// TwinCAT 3 PLC project PLC1
// ProgramVersion: 3.1.4024.0
// libraries:
//   Tc2_Standard, * (Beckhoff Automation GmbH)
//   Tc2_System, * (Beckhoff Automation GmbH)
//   Tc3_Module, * (Beckhoff Automation GmbH)
// project tree:
//   DUTs/ENUM/ E_RS_Cycle_Stop_Cmds.TcDUT, E_Util_State_Cmd.TcDUT, E_TVSA_Cycles.TcDUT, E_Cluster_State_Cmd.TcDUT, E_Util_Service_Req.TcDUT, E_Util_Service_Sts.TcDUT
//   DUTs/STRUCTS/ ST_RS_SeqNumber.TcDUT, ST_Sequence_Sts.TcDUT, ST_Service_Assigned_Sts.TcDUT, ST_Util_Service_Sts.TcDUT, ST_Util_Service_Req.TcDUT
//   DUTs/UNIONS/ U_SeqStart.TcDUT
//   Functions/ F_Get_Seq_Status.TcPOU
//   Function_Blocks/ FB_Cluster_Control.TcPOU, FB_Service_Dispatcher.TcPOU, FB_ReactorSet.TcPOU, FB_ReactorSet_Control.TcPOU, FB_SetOutput_TwoInputs.TcPOU, FB_Utilities_Control.TcPOU, FB_Utilities_Service.TcPOU, FB_Util_Service_Control.TcPOU
//   GVLs/ CONSTANTS.TcGVL, hmi.TcGVL
//   / PlcTask.TcTTO
//   POUs/ MAIN.TcPOU
// real-time tasks:
//   TASK PlcTask: cycle T#10ms, priority 20, ADS port 350
//   TASK PlcTask1: cycle T#10ms, priority 21, ADS port 351
// I/O:
//   DEVICE Device 1 (EtherCAT Automation Protocol) (disabled), AmsNetId 10.33.70.115.2.1
//     Module1 - Publisher
//     Module1 - Subscriber
// variable links:
//   PLC1/PLC1 Instance <-> Device 1 (EtherCAT Automation Protocol)/Module1 - Publisher
//     PlcTask Outputs/MAIN.cluster_control.fb_rs_control[1].fbRS.out_cooling_pump_sts <-> RS1_Bytes/Outputs/VarData[1]
//     PlcTask Outputs/MAIN.cluster_control.fb_rs_control[1].fbRS.out_cycle_req <-> RS1_Bytes/Outputs/VarData[0]
//     PlcTask Outputs/MAIN.cluster_control.fb_rs_control[1].fbRS.out_deadair_pump_sts <-> RS1_Bytes/Outputs/VarData[2]
//     PlcTask Outputs/MAIN.cluster_control.fb_rs_control[1].fbRS.out_steam_system_sts <-> RS1_Bytes/Outputs/VarData[3]
//   PLC1/PLC1 Instance <-> Device 1 (EtherCAT Automation Protocol)/Module1 - Subscriber
//     PlcTask Inputs/MAIN.cluster_control.fb_rs_control[1].fbRS.in_adsorption_seq_sts <-> RS1_Bytes/Inputs/VarData[0]
//     PlcTask Inputs/MAIN.cluster_control.fb_rs_control[1].fbRS.in_airpress_seq_sts <-> RS1_Bytes/Inputs/VarData[4]
//     PlcTask Inputs/MAIN.cluster_control.fb_rs_control[1].fbRS.in_cooling_seq_sts <-> RS1_Bytes/Inputs/VarData[3]
//     PlcTask Inputs/MAIN.cluster_control.fb_rs_control[1].fbRS.in_desorption_seq_sts <-> RS1_Bytes/Inputs/VarData[2]
//     PlcTask Inputs/MAIN.cluster_control.fb_rs_control[1].fbRS.in_evac_seq_sts <-> RS1_Bytes/Inputs/VarData[1]

CONFIGURATION PLC1
    RESOURCE PLC ON TwinCAT3
        TASK PlcTask(INTERVAL := T#10ms, PRIORITY := 20);
        PROGRAM MAIN WITH PlcTask : MAIN;
    END_RESOURCE
END_CONFIGURATION

// ---- DUTs/ENUM/E_RS_Cycle_Stop_Cmds.TcDUT
{attribute 'qualified_only'}
//{attribute 'strict'}
{attribute 'to_string'}

TYPE E_RS_Cycle_Stop_Cmds :
(
	Clear :=0,
	Stop_Cycle,
	Shutdown_Safe,
	Shutdown_Evac,
	Estop
);
END_TYPE

// ---- DUTs/ENUM/E_Util_State_Cmd.TcDUT
{attribute 'qualified_only'}
//{attribute 'strict'}
{attribute 'to_string'}

TYPE E_Util_State_Cmd :
(
	Idle		:= 0,
	Warmup 		:= 1,
	Activate 	:= 2,
	Shutdown 	:= 3,
	Reset_Fault := 4
);
END_TYPE

// ---- DUTs/ENUM/E_TVSA_Cycles.TcDUT
//{attribute 'qualified_only'}
//{attribute 'strict'}
{attribute 'to_string'}

TYPE E_RS_Cycles :
(
	Idle := 0,
	DeadAirEvac,
	SteamDesorption,
	VacCooling,
	AirRepress,
	Adsorption,
	Estop,
	SafeShutdown,
	Error := 9
);
END_TYPE

// ---- DUTs/ENUM/E_Cluster_State_Cmd.TcDUT
{attribute 'qualified_only'}
//{attribute 'strict'}
{attribute 'to_string'}

TYPE E_Cluster_State_Cmd :
(
	Idle := 0,
	Warmup := 1,
	Cycling := 2,
	Shutdown := 3,
	Reset_Fault := 4
);
END_TYPE

// ---- DUTs/ENUM/E_Util_Service_Req.TcDUT
//{attribute 'qualified_only'}
//{attribute 'strict'}
{attribute 'to_string'}

TYPE E_Util_Service_Req :
(
	Reset_Fault := 0,
	On 			:= 1,
	Off 		:= 2
);
END_TYPE

// ---- DUTs/ENUM/E_Util_Service_Sts.TcDUT
//{attribute 'qualified_only'}
//{attribute 'strict'}
{attribute 'to_string'}

TYPE E_Util_Service_Sts :
(
	PowerUp		:= 0,
	Active		:= 1,
	Running		:= 2,
	Faulted		:= 9
);
END_TYPE

// ---- DUTs/STRUCTS/ST_RS_SeqNumber.TcDUT
{attribute 'qualified_only'}
{attribute 'strict'}
TYPE ST_RS_SeqNumber :
STRUCT
	Idle 			: BIT;
	Adsorption		: BIT;
	DeadAirEvac 	: BIT;
	SteamDesorption : BIT;
	VacCooling		: BIT;
	AirRepress 		: BIT;
	Error 			: BIT;
END_STRUCT
END_TYPE

// ---- DUTs/STRUCTS/ST_Sequence_Sts.TcDUT
TYPE ST_Sequence_Sts :
STRUCT
	not_started : BIT;
	started		: BIT;
	completed	: BIT;
	error		: BIT;
END_STRUCT
END_TYPE

// ---- DUTs/STRUCTS/ST_Service_Assigned_Sts.TcDUT
TYPE ST_Service_Assigned_Sts :
STRUCT
	rs_number : UINT;
	is_assigned : BOOL;
END_STRUCT
END_TYPE

// ---- DUTs/STRUCTS/ST_Util_Service_Sts.TcDUT
TYPE ST_Util_Service_Sts :
STRUCT  
	idle		: BOOL;
	ready 		: BOOL;
	running		: BOOL;
	faulted		: BOOL;
	error_code	: DWORD;
END_STRUCT
END_TYPE

// ---- DUTs/STRUCTS/ST_Util_Service_Req.TcDUT
TYPE ST_Util_Service_Req :
STRUCT
	rs_number 		: UINT;
	request_cmd		: UINT;  // (   0 = release/off , 1 = assign/on , 2 =  reset fault)
END_STRUCT
END_TYPE

// ---- DUTs/UNIONS/U_SeqStart.TcDUT
TYPE U_SeqStart :
UNION
	_seq_st 	: ST_RS_SeqNumber;
	_seq_byte 	: BYTE;
END_UNION
END_TYPE

// ---- GVLs/CONSTANTS.TcGVL

VAR_GLOBAL CONSTANT
	rs_count	: UINT := 6;
END_VAR

// ---- GVLs/hmi.TcGVL
{attribute 'qualified_only'}
VAR_GLOBAL
	// Cluster HMI tags - Commnads/Config
	{attribute 'OPC.UA.DA' := '1'} 
	cluster_auto_mode_cmd				: BOOL;
	{attribute 'OPC.UA.DA' := '1'} 								
	cluster_manual_mode_cmd				: BOOL;
	{attribute 'OPC.UA.DA' := '1'} 
	cluster_state_cmd					: BYTE; 									// 0 = Idle, 1 = warmup, 2 = cycle, 3 = shutdown, 4 = reset_fault
	{attribute 'OPC.UA.DA' := '1'} 
	cluster_rs_select_cmd				: ARRAY [1..rs_count] OF BOOL;  			// rs to be started /stopped
	{attribute 'OPC.UA.DA' := '1'} 
	cluster_rs_stop_cycle_cmd			: INT; 										// 1 = stop cycle, 2 = shutdown safe, 3 = shutdown evac, 4 = estop
	{attribute 'OPC.UA.DA' := '1'}  
	cluster_rs_start_cycle_cmd			: BOOL;										// 1 = start cycle
	{attribute 'OPC.UA.DA' := '1'}  
	cluster_reset_fault_cmd				: BOOL;										// reset cluster fault
	{attribute 'OPC.UA.DA' := '1'} 
	cluster_rs_cycles_cfg				: ARRAY [1..rs_count] OF UINT;  			// cycle to run : 12345 = Full TVSA , 1 = Evac, 2 = Desorp ,3 = Cooling ,4 = Repres ,5 = Adsorp
	{attribute 'OPC.UA.DA' := '1'} 
	clsuter_rs_number_of_cycles_cfg		: ARRAY [1..rs_count] OF UINT;  			// number of cycles to run 
	
	// Cluster HMI Tags - Status
	{attribute 'OPC.UA.DA' := '1'} 
	cluster_rs_control_active_cycle_sts : ARRAY [1..rs_count] OF STRING;
	{attribute 'OPC.UA.DA' := '1'} 
	cluster_active_state_sts			: STRING;

	// Utilities HMI tags
	{attribute 'OPC.UA.DA' := '1'} 
	util_auto_mode_cmd		: BOOL := TRUE;  // TRUE = auto mode, FALSE = manual mode 
	{attribute 'OPC.UA.DA' := '1'}  
	util_cooling_pump_cmd 	: REAL; // 0 = off, 1 = On , 2 = reset_fault
	{attribute 'OPC.UA.DA' := '1'} 
	util_cooling_pump_sts 	: INT;
	{attribute 'OPC.UA.DA' := '1'}  
	util_dead_air_pump_cmd 	: REAL; // 0 = off, 1 = On , 2 = reset_fault
	{attribute 'OPC.UA.DA' := '1'} 
	util_dead_air_pump_sts 	: INT;
	{attribute 'OPC.UA.DA' := '1'}  
	util_steam_system_cmd 	: REAL; // 0 = off, 1 = On , 2 = reset_fault
	{attribute 'OPC.UA.DA' := '1'} 
	util_steam_system_sts 	: INT;
	{attribute 'OPC.UA.DA' := '1'}  
	util_purge_assist_cmd 	: REAL; // 0 = off, 1 = On , 2 = reset_fault
	{attribute 'OPC.UA.DA' := '1'} 
	util_purge_assist_sts 	: INT;
END_VAR

// ---- POUs/MAIN.TcPOU
PROGRAM MAIN
VAR
	cluster_control : FB_Cluster_Control();
	sita_out : REAL;
	sita_in1 : REAL;
	sita_in2 : REAL;
	sita_setout : FB_SetOutput_TwoInputs();
END_VAR

cluster_control();

//sita_out := F_SetOutput_LatestInput(in1 := TO_REAL(sita_in1),in2 := TO_REAL(sita_in2));


sita_setout(io_in1 := sita_in1,io_in2 := sita_in2, o_set_value => sita_out);

END_PROGRAM

// ---- Function_Blocks/FB_Cluster_Control.TcPOU
FUNCTION_BLOCK FB_Cluster_Control
VAR
	fb_rs_control 			: ARRAY[1..rs_count] OF FB_ReactorSet_Control;
	//fb_reactor_set			: ARRAY[1..rs_count] OF FB_ReactorSet;
	rs_error				: BOOL;
	
	fb_utilities_control 	: FB_Utilities_Control;
	
	idx_rs 					: UINT;
	
	{attribute 'to_string'}
	seq_state				: (Idle := 0, Warmup := 1, Ready := 2, Cycling := 3, Shutdown := 4, Error); 
	
	rs_stop_cycle_cmd		: ARRAY[1..rs_count] OF  INT;  
	rs_start_cycle_cmd 		: ARRAY[1..rs_count] OF BOOL;
	
	shutdown_util_cmd		: BOOL;
	
	seq_sts 				: ST_Sequence_Sts;
	
	error_reset_cmd			: BOOL;
	trigger_error_reset		: R_TRIG;
	
	cluster_auto_mode		: BOOL;
END_VAR

// Cluster Shutdown 
IF hmi.cluster_state_cmd = E_Cluster_State_Cmd.Shutdown THEN 
	IF  seq_state =  Cycling AND Get_RS_CycleDone_Sts() THEN 
		seq_state := Shutdown;
	ELSIF seq_state <>  Cycling THEN 
		seq_state := Shutdown;
	END_IF
END_IF


// Cluster States 
CASE seq_state OF 
	
	Idle : 
		fb_utilities_control.i_state_req := E_Cluster_State_Cmd.Idle;
		seq_sts.error := FALSE;
		seq_sts.started := FALSE;
		IF hmi.cluster_state_cmd = E_Cluster_State_Cmd.Warmup THEN 
			seq_sts.completed := FALSE;
			seq_sts.started := TRUE;
			seq_state := Warmup;
		END_IF
		
	Warmup:	
		fb_utilities_control.i_state_req := E_Util_State_Cmd.Warmup;
		IF NOT fb_utilities_control.o_bop_warmup_sts.error  THEN 
			IF fb_utilities_control.o_bop_warmup_sts.completed THEN 
				seq_state := Ready;
			END_IF
		ELSE
			seq_state := Error;
		END_IF		
		
	Ready :
		fb_utilities_control.i_state_req := E_Util_State_Cmd.Activate;
		
		IF  NOT fb_utilities_control.o_bop_error_critical AND NOT rs_error THEN
			IF  fb_utilities_control.o_bop_activate_sts.completed AND hmi.cluster_state_cmd = E_Cluster_State_Cmd.Cycling THEN 
				seq_state := Cycling;
			END_IF
		ELSE
			seq_state := Error;
		END_IF
		
	Cycling :
	
			seq_state := Cycling;
		
	Shutdown : 
		
		fb_utilities_control.i_state_req := E_Util_State_Cmd.Shutdown;
		IF NOT fb_utilities_control.o_bop_shutdown_sts.error THEN 
			IF fb_utilities_control.o_bop_shutdown_sts.completed THEN 
				seq_sts.completed := TRUE;
				seq_state := Idle;
			END_IF
		ELSE
			seq_state := Error;	
		END_IF
	
	Error : 
		seq_sts.completed := TRUE;
		seq_sts.error := TRUE;
		IF error_reset_cmd THEN 
			seq_state := Idle;
		END_IF		
END_CASE


// Reactor Sets and Utilities Cycles Control 
RS_Utilities_Control();

// Error Reset Handling 
Reset_Error();

// ==============  HMI ===================

// HMI auto/manual
IF hmi.cluster_auto_mode_cmd THEN 
	cluster_auto_mode := TRUE;
	hmi.cluster_auto_mode_cmd := FALSE;
ELSIF hmi.cluster_manual_mode_cmd THEN 
	cluster_auto_mode := FALSE;
	hmi.cluster_manual_mode_cmd := FALSE;
END_IF

// Cycle Stauts to HMI 
FOR idx_rs := 1 TO rs_count DO
	hmi.cluster_rs_control_active_cycle_sts[idx_rs] := TO_STRING(fb_rs_control[idx_rs].Active_Cycle);	
END_FOR
hmi.cluster_active_state_sts := TO_STRING(seq_state);

METHOD Get_RS_CycleDone_Sts : BOOL
VAR
	rs_done : BOOL;
END_VAR
rs_done := fb_rs_control[1].o_Done;
FOR idx_rs := 2 TO rs_count DO 
	rs_done := rs_done AND fb_rs_control[idx_rs].o_Done;
END_FOR
Get_RS_CycleDone_Sts := rs_done;
END_METHOD

METHOD Get_RS_ServiceAssiged_Sts : BOOL
VAR_INPUT
	i_rs_number : UINT;
	i_assigned_rs_list : ARRAY[1..rs_count] OF UINT; 
END_VAR
VAR
	idx_rs : UINT;
END_VAR
// TRUE if the RS is assigned to an utilities service 

FOR idx_rs := 1 TO rs_count DO 
	IF i_rs_number = i_assigned_rs_list[idx_rs] THEN
		Get_RS_ServiceAssiged_Sts := TRUE;
		EXIT;
	END_IF
END_FOR
END_METHOD

METHOD Reset_Error : BOOL
VAR_INPUT
END_VAR

fb_utilities_control.i_fault_reset := hmi.cluster_reset_fault_cmd ;
FOR idx_rs := 1 TO rs_count DO 
//	fb_reactor_set[idx_rs].i_fault_reset := hmi.cluster_reset_fault_cmd;
	fb_rs_control[idx_rs].i_reset_fault  := hmi.cluster_reset_fault_cmd;
END_FOR
hmi.cluster_reset_fault_cmd := FALSE;
END_METHOD

ACTION RS_Utilities_Control:
StartStop_RS_Cycle();

FOR idx_rs := 1 TO rs_count DO 	
	
	fb_rs_control[idx_rs]( 	i_rs_number				:= idx_rs,
							io_cycle_selection 		:= hmi.cluster_rs_cycles_cfg[idx_rs],
							io_cycles_number_to_run := hmi.clsuter_rs_number_of_cycles_cfg[idx_rs],
							io_start_cycle 			:= rs_start_cycle_cmd[idx_rs],						
							io_stop_cycle 			:= rs_stop_cycle_cmd[idx_rs],
							i_cooling_pump_assigned := Get_RS_ServiceAssiged_Sts(i_rs_number := idx_rs, i_assigned_rs_list := fb_utilities_control.cooling_pump.assigned_rs_number),
							i_cooling_pump_sts 		:= fb_utilities_control.cooling_pump.o_service_sts,
							i_deadair_pump_assigned	:= Get_RS_ServiceAssiged_Sts(i_rs_number := idx_rs, i_assigned_rs_list := fb_utilities_control.dead_air_pump.assigned_rs_number),
							i_deadair_pump_sts 		:= fb_utilities_control.dead_air_pump.o_service_sts,
							i_steam_system_assigned	:= Get_RS_ServiceAssiged_Sts(i_rs_number := idx_rs, i_assigned_rs_list := fb_utilities_control.steam_sytem.assigned_rs_number),
							i_steam_system_sts 		:= fb_utilities_control.steam_sytem.o_service_sts,
							i_purge_assist_assigned := Get_RS_ServiceAssiged_Sts(i_rs_number := idx_rs, i_assigned_rs_list := fb_utilities_control.purge_assist.assigned_rs_number),
							i_purge_assist_sts 		:= fb_utilities_control.purge_assist.o_service_sts,
							o_cooling_pump_req		=> fb_utilities_control.i_cooling_pump_req,
							o_deadair_pump_req		=> fb_utilities_control.i_deadair_pump_req,
							o_steam_system_req		=> fb_utilities_control.i_steam_system_req,
							o_purge_assist_req		=> fb_utilities_control.i_purge_assist_req);
							
	fb_utilities_control(i_rs_number_service_req := idx_rs);	
			
END_FOR

fb_utilities_control.State_Control();
END_ACTION

METHOD StartStop_RS_Cycle : BOOL
VAR
	idx_rs 				: UINT;
END_VAR
// HMI Start Commands
IF hmi.cluster_rs_start_cycle_cmd THEN
   IF cluster_auto_mode THEN 
		FOR idx_rs := 1 TO rs_count DO
			IF NOT fb_rs_control[idx_rs].o_Started AND NOT fb_rs_control[idx_rs].o_Error THEN
				rs_start_cycle_cmd[idx_rs] := TRUE;
			END_IF
		END_FOR
	END_IF
	hmi.cluster_rs_start_cycle_cmd := FALSE;
	hmi.cluster_rs_stop_cycle_cmd := 0;
END_IF



// Reactor Set Errors Stop Commands Requests  + HMI Stop req ( auto mode only) 
IF cluster_auto_mode THEN 
	FOR idx_rs := 1 TO rs_count DO
		IF NOT fb_rs_control[idx_rs].o_Stopping THEN 
			IF fb_rs_control[idx_rs].fbRS.o_error_estop_req OR fb_utilities_control.o_bop_error_critical THEN   // RS error  + BOP Error -> Estop Request 
				rs_stop_cycle_cmd[idx_rs] := E_RS_Cycle_Stop_Cmds.Estop;
			ELSIF fb_rs_control[idx_rs].fbRS.o_error_shutdown_req THEN
				rs_stop_cycle_cmd[idx_rs] := E_RS_Cycle_Stop_Cmds.Shutdown_Safe;			// RS errror -> Shutdown Safe Req
			ELSIF hmi.cluster_rs_stop_cycle_cmd > 0 THEN
				rs_stop_cycle_cmd[idx_rs] := hmi.cluster_rs_stop_cycle_cmd;					// HMI Request 
			ELSE
				rs_stop_cycle_cmd[idx_rs] := E_RS_Cycle_Stop_Cmds.Clear;
			END_IF
		END_IF
	END_FOR
END_IF


// HMI Stop Command (Cycle Stop, Shutdown, Shutdown Evac, Estop) 
IF hmi.cluster_rs_stop_cycle_cmd > 0  THEN
	hmi.cluster_rs_stop_cycle_cmd := 0;
	hmi.cluster_rs_start_cycle_cmd := FALSE;
END_IF
END_METHOD

END_FUNCTION_BLOCK

// ---- Function_Blocks/FB_ReactorSet_Control.TcPOU
FUNCTION_BLOCK FB_ReactorSet_Control
VAR_IN_OUT
	io_stop_cycle 			: INT;
	io_cycle_selection		: UINT;  // 12345 = Full TVSA Cycle , 1 = Evac , 2 = Desorp , 3 = Cooling, 4 = Repres, 5 = Adsorp
	io_cycles_number_to_run	: UINT;	
	io_start_cycle 			: BOOL;
END_VAR

VAR_INPUT
	i_rs_number 				: UINT;
	i_start_cycle_adsorption	: BOOL;
	i_reset_fault				: BOOL;

	//Utilities Services Status
	i_cooling_pump_sts 		: ST_Util_Service_Sts;
	i_deadair_pump_sts 		: ST_Util_Service_Sts;
	i_steam_system_sts 		: ST_Util_Service_Sts;
	i_purge_assist_sts		: ST_Util_Service_Sts;	
	i_cooling_pump_assigned : BOOL;
	i_deadair_pump_assigned	: BOOL;
	i_steam_system_assigned	: BOOL;
	i_purge_assist_assigned	: BOOL;
	
END_VAR
VAR_OUTPUT
	o_Error 				: BOOL;
	o_Started 				: BOOL;
	o_Done 					: BOOL;
	o_Stopping				: BOOL;
	
	// RS to Utilities Request
	o_cooling_pump_req		: BYTE;  
	o_deadair_pump_req		: BYTE;
	o_steam_system_req		: BYTE;
	o_purge_assist_req		: BYTE;
END_VAR
VAR

	cycle_state 				: E_RS_Cycles := Idle;
	cycles_to_run 				: UINT;
	cycles_completed			: UINT := 0 ;
	trig_start_cmd				: R_TRIG;
	cycle_first_entry			: BOOL;
	trig_cycle_first_run		: R_TRIG;
	cycle_single_selected		: BOOL;
	
	trig_stop_cmd				: R_TRIG;
	shutdown_evac_req			: BOOL := FALSE;
	fbRS						: FB_ReactorSet;
	
	adsorption_seq_sts 		: ST_Sequence_Sts;
	evac_seq_sts 			: ST_Sequence_Sts;
	desorption_seq_sts 		: ST_Sequence_Sts;
	cooling_seq_sts 		: ST_Sequence_Sts;
	airpress_seq_sts 		: ST_Sequence_Sts;
	estop_seq_sts			: ST_Sequence_Sts;
	shutdown_seq_sts		: ST_Sequence_Sts;
	
	rs_error_active			: BOOL;
	
END_VAR


// State Machine
 
CycleStart_Handler();


CASE cycle_state OF 
	
	Idle: 
		 CycleEntry_Handler(i_current_state := Idle);
		 
		 o_Started := FALSE;
		 o_Error := FALSE;	
		 cycles_to_run := 0;	
		 
	DeadAirEvac :
		CycleEntry_Handler(i_current_state := DeadAirEvac);
		IF NOT evac_seq_sts.error THEN 	
			IF evac_seq_sts.completed THEN
				CycleNext_Handler(i_current_state := DeadAirEvac);	
			END_IF
		ELSE
			CycleError_Handler();
		END_IF
	
	SteamDesorption : 
		CycleEntry_Handler(i_current_state := SteamDesorption);
		IF NOT desorption_seq_sts.error THEN 	
			IF desorption_seq_sts.completed THEN
				CycleNext_Handler(i_current_state := SteamDesorption);	
			END_IF
		ELSE
			CycleError_Handler();
		END_IF
	
	VacCooling: 
		CycleEntry_Handler(i_current_state := VacCooling);
		IF NOT cooling_seq_sts.error THEN 	
			IF cooling_seq_sts.completed THEN
				CycleNext_Handler(i_current_state := VacCooling);	
			END_IF
		ELSE
			CycleError_Handler();
		END_IF
	
	AirRepress :
		CycleEntry_Handler(i_current_state := AirRepress);
		IF NOT airpress_seq_sts.error THEN 	
			IF airpress_seq_sts.completed THEN
				CycleNext_Handler(i_current_state := AirRepress);			
			END_IF
		ELSE
			CycleError_Handler();
		END_IF
		
			
	Adsorption :
		CycleEntry_Handler(i_current_state := Adsorption);
		IF NOT adsorption_seq_sts.error THEN 	
			IF adsorption_seq_sts.completed THEN
				CycleNext_Handler(i_current_state := Adsorption);	
			END_IF
		ELSE
			CycleError_Handler();
		END_IF
		
	
	Estop : 		
		CycleEntry_Handler(i_current_state := Estop);
		IF NOT estop_seq_sts.error THEN 	
			IF estop_seq_sts.completed THEN
				CycleNext_Handler(i_current_state := Estop);			
			END_IF
		ELSE
			CycleError_Handler();
		END_IF
		
	SafeShutdown : 		
		CycleEntry_Handler(i_current_state := SafeShutdown);
		IF NOT shutdown_seq_sts.error THEN 	
			IF shutdown_seq_sts.completed THEN
				CycleNext_Handler(i_current_state := SafeShutdown);
				shutdown_evac_req := FALSE;			
			END_IF
		ELSE
			CycleError_Handler();
		END_IF
		
	Error : 
		CycleEntry_Handler(i_current_state := Error);
		o_Error := TRUE;
		o_Done := TRUE;
		o_Started := FALSE;
		shutdown_evac_req := FALSE;
		IF i_reset_fault THEN 
			CycleNext_Handler(i_current_state := Error);	
		END_IF

END_CASE


CycleStop_Handler();

// Reactor Set IOs Control 

fbRS(i_cycle_req 				:= active_cycle,
	 i_fault_reset				:= i_reset_fault,
	 i_cooling_pump_assigned 	:= i_cooling_pump_assigned,
	 i_cooling_pump_sts 		:= i_cooling_pump_sts,
	 i_deadair_pump_assigned	:= i_deadair_pump_assigned,
	 i_deadair_pump_sts 		:= i_deadair_pump_sts,
	 i_steam_system_assigned	:= i_steam_system_assigned,
	 i_steam_system_sts 		:= i_steam_system_sts,
	 i_purge_assist_assigned 	:= i_purge_assist_assigned,
	 i_purge_assist_sts 		:= i_purge_assist_sts,
	 o_adsorption_seq_sts 		=> adsorption_seq_sts,
	 o_airpress_seq_sts			=> airpress_seq_sts,
	 o_evac_seq_sts 			=> evac_seq_sts,
	 o_desorption_seq_sts 		=> desorption_seq_sts,
	 o_cooling_seq_sts			=> cooling_seq_sts,
	 o_estop_seq_sts			=> estop_seq_sts,
	 o_shutdown_seq_sts			=> shutdown_seq_sts,
	 o_cooling_pump_req			=> o_cooling_pump_req,
	 o_deadair_pump_req			=> o_deadair_pump_req,
	 o_steam_system_req			=> o_steam_system_req,
	 o_purge_assist_req			=> o_purge_assist_req,
	 o_error_active				=> rs_error_active );

PROPERTY active_cycle : E_RS_Cycles
GET
active_cycle := cycle_state;
END_GET
END_PROPERTY

METHOD CycleEntry_Handler : BOOL
VAR_INPUT
	i_current_state : E_RS_Cycles;
END_VAR
trig_cycle_first_run(CLK := cycle_first_entry) ;
cycle_first_entry := TRUE;
IF trig_cycle_first_run.Q THEN 
	Logger();
END_IF
END_METHOD

METHOD CycleError_Handler : BOOL
VAR_INPUT
END_VAR
cycle_first_entry := FALSE;
trig_cycle_first_run(CLK := cycle_first_entry) ;
cycle_state := Error;
END_METHOD

METHOD PRIVATE CycleNext_Handler : INT
VAR_INPUT
	i_current_state : E_RS_Cycles;
END_VAR
// single cycle selected 
IF (i_current_state = Estop) OR  (i_current_state = SafeShutdown) THEN 
	o_Done := TRUE;
	cycle_state := Idle; 
ELSIF cycle_single_selected THEN 
	o_Done := TRUE;
	cycle_state := Idle; 
	cycle_single_selected := FALSE;
// tvsa cycle complete 
ELSIF ((i_current_state = Adsorption) AND (cycles_completed = cycles_to_run))  THEN 
	o_Done := TRUE;
	cycle_state := Idle;
// next tvsa cycle
ELSIF (i_current_state = Adsorption)  AND (cycles_completed < cycles_to_run )  THEN 
	cycle_state := DeadAirEvac ;
	cycles_completed := cycles_completed + 1;
// next state/cycle
ELSIF (NOT (i_current_state = Adsorption)) AND  (NOT (i_current_state = Error)) THEN
	cycle_state := i_current_state + 1;
ELSIF (i_current_state = DeadAirEvac) AND shutdown_evac_req THEN 
	cycle_state := SafeShutdown; 	
ELSIF i_current_state = Error THEN
	o_Error := FALSE;
	cycle_state := Idle ;	
END_IF

cycle_first_entry := FALSE;
//trig_cycle_first_run(CLK := cycle_first_entry) ;
END_METHOD

ACTION CycleStart_Handler:

trig_start_cmd(CLK := io_start_cycle = TRUE);

IF trig_start_cmd.Q THEN 

	IF ( io_cycle_selection = 0 OR io_cycles_number_to_run = 0 ) AND NOT (cycle_state = Error) THEN 
		cycle_single_selected := FALSE;	
		cycle_state := Idle;
	ELSIF io_cycle_selection = 12345 THEN
		cycles_to_run := io_cycles_number_to_run;
//		cycle_first_entry := FALSE;
		cycle_single_selected := FALSE;	
		IF i_start_cycle_adsorption THEN 
			cycle_state := Adsorption; 
		ELSE
			cycle_state := DeadAirEvac;
		END_IF
	ELSIF io_cycle_selection >= 1 AND io_cycle_selection <=5 THEN
		cycle_single_selected := TRUE;
		cycle_state := TO_INT(io_cycle_selection);
	END_IF
	
	o_Done := FALSE;
	o_Started := TRUE;
	o_Error := FALSE;
	
	cycle_first_entry := FALSE;
	cycles_completed := 0 ;
	
	io_cycle_selection := 0;
	io_cycles_number_to_run := 0;
	io_start_cycle := FALSE;
	
END_IF
END_ACTION

ACTION CycleStop_Handler:
trig_stop_cmd( CLK := io_stop_cycle > 0);
IF trig_stop_cmd.Q THEN 
	IF io_stop_cycle = E_RS_Cycle_Stop_Cmds.Stop_Cycle THEN 
		cycles_to_run := cycles_completed + 1 ;	
	ELSIF io_stop_cycle = E_RS_Cycle_Stop_Cmds.Shutdown_Safe THEN 
		cycle_state := SafeShutdown;
	ELSIF io_stop_cycle = E_RS_Cycle_Stop_Cmds.Shutdown_Evac THEN 
		shutdown_evac_req := TRUE;
		cycle_state := DeadAirEvac;
	ELSIF io_stop_cycle = E_RS_Cycle_Stop_Cmds.Estop THEN 
		cycle_state := Estop;
	END_IF
	io_stop_cycle := 0;
END_IF

o_Stopping := cycle_state = Estop OR cycle_state = SafeShutdown;
END_ACTION

METHOD Logger : BOOL
VAR_INPUT
END_VAR
ADSLOGSTR(msgCtrlMask := ADSLOG_MSGTYPE_WARN,msgFmtStr := 'Reactor Set : %s' ,strArg := TO_STRING(i_rs_number));
ADSLOGSTR(msgCtrlMask := ADSLOG_MSGTYPE_WARN,msgFmtStr := 'Sequence : %s' ,strArg := TO_STRING(cycle_state));
ADSLOGSTR(msgCtrlMask := ADSLOG_MSGTYPE_WARN,msgFmtStr := 'Cycle Number : %s' ,strArg := TO_STRING(cycles_completed));
END_METHOD

END_FUNCTION_BLOCK

// ---- Function_Blocks/FB_ReactorSet.TcPOU
FUNCTION_BLOCK FB_ReactorSet
VAR_INPUT
	i_cycle_req 			: E_RS_Cycles;
	i_cooling_pump_sts 		: ST_Util_Service_Sts;
	i_deadair_pump_sts 		: ST_Util_Service_Sts;
	i_steam_system_sts 		: ST_Util_Service_Sts;
	i_purge_assist_sts		: ST_Util_Service_Sts;	
	i_cooling_pump_assigned : BOOL;
	i_deadair_pump_assigned	: BOOL;
	i_steam_system_assigned	: BOOL;
	i_purge_assist_assigned	: BOOL;
	i_fault_reset			: BOOL;
	
END_VAR
VAR_OUTPUT
	o_adsorption_seq_sts 	: ST_Sequence_Sts;
	o_evac_seq_sts 			: ST_Sequence_Sts;
	o_desorption_seq_sts 	: ST_Sequence_Sts;
	o_cooling_seq_sts 		: ST_Sequence_Sts;
	o_airpress_seq_sts 		: ST_Sequence_Sts;
	o_estop_seq_sts 		: ST_Sequence_Sts;
	o_shutdown_seq_sts 		: ST_Sequence_Sts;
	
	o_cooling_pump_req		: BYTE;  
	o_deadair_pump_req		: BYTE;
	o_steam_system_req		: BYTE;
	o_purge_assist_req		: BYTE;
	
	o_error_active				: BOOL;
	o_error_code				: DWORD;
	o_error_code_evac			: DWORD;
	o_error_code_desorption		: DWORD;
	o_error_code_cooling		: DWORD;
	o_error_code_repress		: DWORD;
	o_error_code_adsorption		: DWORD;
	
	o_error_shutdown_req		: BOOL;
	o_error_estop_req			: BOOL;
	
	
END_VAR
VAR
	
	// from RS Controller 
	in_adsorption_seq_sts  	AT %I*	: BYTE;
	in_evac_seq_sts 		AT %I*	: BYTE;
	in_desorption_seq_sts 	AT %I*	: BYTE;
	in_cooling_seq_sts 		AT %I*	: BYTE;
	in_airpress_seq_sts 	AT %I*	: BYTE;
	in_estop_seq_sts 		AT %I*	: BYTE;
	in_shutdown_seq_sts 	AT %I*	: BYTE;
	
	in_cooling_pump_req		AT %I*	: BYTE;  
	in_deadair_pump_req		AT %I*	: BYTE;
	in_steam_system_req		AT %I*	: BYTE;
	in_purge_assist_req		AT %I*	: BYTE;
	
	in_error_sts			AT %I* 	: BOOL;
	in_error_code1			AT %I*	: DWORD;
	in_error_code2			AT %I*	: DWORD;
	
	in_error_shutdown_req	AT %I* : BOOL;
	in_error_estop_req		AT %I* : BOOL;
	
	
	
	// to RS Controller
	out_cycle_req 				AT %Q*	: BYTE;
	
	out_cooling_pump_sts 		AT %Q*	: BYTE;  
	out_deadair_pump_sts		AT %Q*	: BYTE;
	out_steam_system_sts		AT %Q*	: BYTE;
	out_purge_assist_sts		AT %Q*	: BYTE;
	
	out_cooling_pump_assigned 		AT %Q* : BOOL;
	out_deadair_pump_assigned		AT %Q*: BOOL;
	out_steam_system_assigned		AT %Q*: BOOL;
	out_purge_assist_assigned		AT %Q*: BOOL;
	
	out_error_reset					AT %Q* : BOOL;
		
	
END_VAR

// Sequence Select + Run request to RS controller

out_cycle_req := TO_BYTE(i_cycle_req);

// Fault Reset to RS Controller

out_error_reset := i_fault_reset;

// Service Request Assigned Sts to RS Controller

out_cooling_pump_assigned	:= i_cooling_pump_assigned;
out_deadair_pump_assigned	:= i_deadair_pump_assigned;
out_steam_system_assigned	:= i_steam_system_assigned;
out_purge_assist_assigned	:= i_purge_assist_assigned;

// Utilities Services Status  to RS Copntroller 

Set_Service_Sts ( i_service_sts := i_cooling_pump_sts,o_service_sts => out_cooling_pump_sts);
Set_Service_Sts ( i_service_sts := i_deadair_pump_sts,o_service_sts => out_deadair_pump_sts);
Set_Service_Sts ( i_service_sts := i_steam_system_sts,o_service_sts => out_steam_system_sts);
Set_Service_Sts ( i_service_sts := i_purge_assist_sts,o_service_sts => out_purge_assist_sts);

//

// Seq Status from RS controller 

F_Get_Seq_Status(i_seq_sts := in_adsorption_seq_sts,o_seq_sts => o_adsorption_seq_sts);
F_Get_Seq_Status(i_seq_sts := in_evac_seq_sts,o_seq_sts => o_evac_seq_sts);
F_Get_Seq_Status(i_seq_sts := in_desorption_seq_sts,o_seq_sts => o_desorption_seq_sts);
F_Get_Seq_Status(i_seq_sts := in_cooling_seq_sts,o_seq_sts => o_cooling_seq_sts);
F_Get_Seq_Status(i_seq_sts := in_airpress_seq_sts,o_seq_sts => o_airpress_seq_sts);
F_Get_Seq_Status(i_seq_sts := in_estop_seq_sts,o_seq_sts => o_estop_seq_sts);
F_Get_Seq_Status(i_seq_sts := in_shutdown_seq_sts,o_seq_sts => o_shutdown_seq_sts);

// Utilities Req from RS Controller 

o_cooling_pump_req		:= in_cooling_pump_req;
o_deadair_pump_req		:= in_deadair_pump_req;
o_steam_system_req		:= in_steam_system_req;
o_purge_assist_req		:= in_purge_assist_req;

// Error mapping from RS Controller
o_error_active := in_error_sts;

// Stop Request triggered by RS errors
o_error_shutdown_req := in_error_shutdown_req;
o_error_estop_req := in_error_estop_req;

METHOD Set_Service_Sts : BOOL
VAR_INPUT
	i_service_sts : ST_Util_Service_Sts;
END_VAR
VAR_OUTPUT
	o_service_sts	: BYTE;
END_VAR
IF i_service_sts.ready THEN
	o_service_sts := 1 ;
ELSIF i_service_sts.running THEN
	o_service_sts := 2 ;
ELSIF i_service_sts.faulted THEN
	o_service_sts := 9 ;
ELSE
	o_service_sts := 0 ;	
END_IF
END_METHOD

END_FUNCTION_BLOCK

// ---- Functions/F_Get_Seq_Status.TcPOU
FUNCTION F_Get_Seq_Status : BOOL
VAR_INPUT
	i_seq_sts : BYTE;
END_VAR
VAR_OUTPUT
	o_seq_sts : ST_Sequence_Sts;
END_VAR

o_seq_sts.not_started 		:= i_seq_sts = 0;
o_seq_sts.started 			:= i_seq_sts = 1;
o_seq_sts.completed 		:= i_seq_sts = 2;
o_seq_sts.error 			:= i_seq_sts = 9;

END_FUNCTION

// ---- Function_Blocks/FB_Utilities_Control.TcPOU
FUNCTION_BLOCK FB_Utilities_Control

VAR_INPUT	
	i_state_req				: INT;
	i_fault_reset			: BOOL;
	i_rs_number_service_req	: UINT;
	i_cooling_pump_req		: UINT;
	i_deadair_pump_req		: UINT;
	i_steam_system_req		: UINT;
	i_purge_assist_req		: UINT;	
END_VAR

VAR_OUTPUT
	o_bop_error_critical	: BOOL;
	o_bop_error_warning		: BOOL;
	o_bop_warmup_sts		: ST_Sequence_Sts;
	o_bop_activate_sts		: ST_Sequence_Sts;
	o_bop_shutdown_sts		: ST_Sequence_Sts;
END_VAR

VAR
	
	util_state : ( Idle := 0, Warmup := 1, Active := 2, Shutdown := 3, Error := 4); 
	
	cooling_pump_req		: ST_Util_Service_Req;
	deadair_pump_req		: ST_Util_Service_Req;
	steam_system_req		: ST_Util_Service_Req;
	purge_assist_req		: ST_Util_Service_Req;	
	
	cooling_pump	: FB_Util_Service_Control(shared_rs_count := rs_count, module_rs_constrain := FALSE, manual_control_only := FALSE);
	dead_air_pump	: FB_Util_Service_Control(shared_rs_count := 1,		   module_rs_constrain := FALSE, manual_control_only := FALSE);
	steam_sytem 	: FB_Util_Service_Control(shared_rs_count := 2, 	   module_rs_constrain := TRUE,  manual_control_only := TRUE);
	purge_assist 	: FB_Util_Service_Control(shared_rs_count := rs_count, module_rs_constrain := FALSE, manual_control_only := FALSE);
		
	comms_fault		: BOOL;
	service_fault	: BOOL;
	
	
	// BOP IOs
	
	in_bop_warmup_sts 		AT %I* : BYTE;
	in_bop_activate_sts		AT %I* : BYTE;
	in_bop_shutdown_sts		AT %I* : BYTE;
	in_bop_error			AT %I* : BOOL;
	in_bop_error_code1		AT %I* : DWORD;
	in_bop_error_code2		AT %I* : DWORD;
	

	out_util_state_req 		AT %Q* : INT; // 0 = Idle, 1 = warmup, 2 = activavte, 3 = shutdown 
	out_util_reset_fault	AT %Q* : BOOL;
	
END_VAR


// Services FBds calls

cooling_pump_req.request_cmd := i_cooling_pump_req;
cooling_pump_req.rs_number := i_rs_number_service_req;
cooling_pump( i_service_req := cooling_pump_req, i_manual_service_req := hmi.util_cooling_pump_cmd,i_auto_mode := hmi.util_auto_mode_cmd);

deadair_pump_req.request_cmd := i_deadair_pump_req;
deadair_pump_req.rs_number := i_rs_number_service_req;
dead_air_pump( i_service_req := deadair_pump_req, i_manual_service_req := hmi.util_dead_air_pump_cmd,i_auto_mode := hmi.util_auto_mode_cmd); 

steam_system_req.request_cmd := i_steam_system_req;
steam_system_req.rs_number := i_rs_number_service_req;
steam_sytem( i_service_req := steam_system_req, i_manual_service_req := hmi.util_steam_system_cmd,i_auto_mode := hmi.util_auto_mode_cmd); 
//steam_sytem( i_manual_service_req := hmi.util_steam_system_cmd,i_auto_mode := hmi.util_auto_mode_cmd,i_auto_mode := hmi.util_auto_mode_cmd); 

purge_assist_req.request_cmd := i_purge_assist_req;
purge_assist_req.rs_number := i_rs_number_service_req;
purge_assist( i_service_req := purge_assist_req, i_manual_service_req := hmi.util_purge_assist_cmd); 

// IOs parsing 

GetSet_BOP_IOs();

// Erros Handling 

o_bop_error_critical := in_bop_error AND in_bop_error_code1.0 AND in_bop_error_code2.3 ; // TBD for adding more erros to the list of critical errors 
o_bop_error_warning  := in_bop_error AND in_bop_error_code1.1 AND in_bop_error_code2.1 ; // TBD to add more errors to the list of warnings 

service_fault := cooling_pump.o_service_sts.faulted OR dead_air_pump.o_service_sts.faulted OR steam_sytem.o_service_sts.faulted OR purge_assist.o_service_sts.faulted ;

METHOD GetSet_BOP_IOs : BOOL
VAR_INPUT
END_VAR

// Get IOs

F_Get_Seq_Status( i_seq_sts := in_bop_warmup_sts, o_seq_sts => o_bop_warmup_sts);
F_Get_Seq_Status( i_seq_sts := in_bop_activate_sts, o_seq_sts => o_bop_activate_sts);
F_Get_Seq_Status( i_seq_sts := in_bop_shutdown_sts, o_seq_sts => o_bop_shutdown_sts);
END_METHOD

METHOD State_Control : BOOL
VAR_INPUT
END_VAR
IF i_state_req = E_Util_State_Cmd.Shutdown THEN
	util_state := Shutdown;
END_IF

IF in_bop_error OR service_fault THEN
	util_state := Error;
END_IF



CASE util_state OF 
	
	Idle : 
		IF i_state_req = E_Util_State_Cmd.Warmup  AND NOT in_bop_error THEN 
			util_state := Warmup;
		ELSIF 	in_bop_error THEN 
			util_state := Error;
		END_IF
	Warmup: 
		out_util_state_req := Warmup;
		IF NOT o_bop_warmup_sts.error THEN 
			IF o_bop_warmup_sts.completed AND i_state_req = E_Util_State_Cmd.Activate THEN 
				util_state := Active;
			END_IF
		ELSE
			util_state := Error;
		END_IF
	Active: 
		out_util_state_req := E_Util_Service_Sts.Active;
		IF  o_bop_activate_sts.error THEN 
			util_state := Error;
		END_IF
		
	Shutdown : 
		out_util_state_req := Shutdown;
		IF NOT o_bop_shutdown_sts.error THEN 
			IF o_bop_shutdown_sts.completed THEN 
				util_state := Idle;
			END_IF
		ELSE
			util_state := Error;
		END_IF
	Error: 
		cooling_pump.Clear_RS_Queue();
		dead_air_pump.Clear_RS_Queue();
		steam_sytem.Clear_RS_Queue();
		purge_assist.Clear_RS_Queue();	
		IF i_fault_reset THEN 
			out_util_reset_fault := TRUE;
			IF NOT in_bop_error THEN
				util_state := Idle;
			END_IF
		END_IF
		
END_CASE
END_METHOD

END_FUNCTION_BLOCK

// ---- Function_Blocks/FB_Util_Service_Control.TcPOU
FUNCTION_BLOCK FB_Util_Service_Control

VAR_INPUT
	i_service_req			: ST_Util_Service_Req;
	i_manual_service_req	: REAL;	
	i_auto_mode				: BOOL;
END_VAR

VAR_OUTPUT
	o_service_sts 			: ST_Util_Service_Sts;
END_VAR

VAR
	shared_rs_count  		: UINT;     // max number of rs to be assigned to the util service
	module_rs_constrain		: BOOL;		// same module assignment constrain
	manual_control_only		: BOOL;		// manual control only 
	
	service_req 			: REAL;
	service_req_dispatcher	: BOOL;
		
	fb_dispatcher 			: FB_Service_Dispatcher;
	
	fb_service_cmd 			: FB_SetOutput_TwoInputs ;
	
	// IOs to Utilities PLC
	in_service_sts 			AT %I* : BYTE;
	in_service_error_code  	AT %I* : DWORD;
		
	out_service_req 		AT %Q* : BYTE;
END_VAR


IF o_service_sts.faulted THEN 
	fb_dispatcher.Clear_Queue();
	service_req := 0;
ELSE
	IF manual_control_only THEN 
		fb_dispatcher( i_service_req := i_service_req,i_shared_rs := shared_rs_count, i_rs_module_constrain := module_rs_constrain, o_service_req => service_req_dispatcher);
		service_req := i_manual_service_req;
	ELSE
		IF i_auto_mode THEN
			// manage the rs assignment queue based on request form reactor set controller, max number of RSs shared by the service and the number of RSs whithin the same module that can sahre the same service 
			fb_dispatcher( i_service_req := i_service_req,i_shared_rs := shared_rs_count, i_rs_module_constrain := module_rs_constrain, o_service_req => service_req_dispatcher);
			service_req := TO_REAL(service_req_dispatcher);
		ELSE
			fb_dispatcher.Clear_Queue();
			service_req := i_manual_service_req;
		END_IF
	END_IF
END_IF

IOs_Mapping();

PROPERTY assigned_rs_number : ARRAY[1..rs_count] OF UINT
GET
assigned_rs_number := fb_dispatcher.o_assigned_rs_number;
END_GET
END_PROPERTY

METHOD Clear_RS_Queue : BOOL
fb_dispatcher.Clear_Queue();
END_METHOD

METHOD FB_init : BOOL
VAR_INPUT
	bInitRetains 		: BOOL; // if TRUE, the retain variables are initialized (warm start / cold start)
	bInCopyCode 		: BOOL;  // if TRUE, the instance afterwards gets moved into the copy code (online change)
	shared_rs_count  	: UINT;
	module_rs_constrain	: BOOL;
	manual_control_only : BOOL;
END_VAR
THIS^.shared_rs_count := shared_rs_count;
THIS^.module_rs_constrain := module_rs_constrain;
THIS^.manual_control_only := manual_control_only;
END_METHOD

METHOD IOs_Mapping : BOOL
VAR_INPUT
END_VAR
out_service_req := TO_BYTE(service_req);


o_service_sts.idle 			:= in_service_sts = E_Util_Service_Sts.PowerUp;
o_service_sts.ready 		:= in_service_sts = E_Util_Service_Sts.Active;
o_service_sts.running 		:= in_service_sts = E_Util_Service_Sts.Running;
o_service_sts.faulted 		:= in_service_sts = E_Util_Service_Sts.Faulted;
o_service_sts.error_code	:= in_service_error_code;
END_METHOD

END_FUNCTION_BLOCK

// ---- Function_Blocks/FB_Service_Dispatcher.TcPOU
FUNCTION_BLOCK FB_Service_Dispatcher
VAR_INPUT
	i_service_req 			: ST_Util_Service_Req;
	i_shared_rs 			: UINT;		  // max number of reactor sets  the util service can be shared by 
	i_rs_module_constrain  	: BOOL;       // true if the reactors sets cannot be par of the same module
END_VAR
VAR_OUTPUT
	o_service_req			: BOOL;  // on/off request to utilities 
	o_assigned_rs_number	: ARRAY[1..rs_count] OF UINT; // rs number that has been assigned to a service 
END_VAR
VAR
	service_req_queue		: ARRAY [1..rs_count] OF ST_Service_Assigned_Sts;
	idx_queue				: UINT;
	idx_queue_update		: UINT;
	trig_service_assign		: R_TRIG;
	trig_service_release	: R_TRIG;
	
	service_assign			: BOOL;
	service_release			: BOOL;
	
	rs_same_module			: BOOL;
END_VAR

// Add to queue 

FOR idx_queue := 1 TO rs_count DO
	IF (i_service_req.request_cmd = TO_UINT(E_Util_Service_Req.On))  THEN 
		IF  (service_req_queue[idx_queue].rs_number = i_service_req.rs_number)  THEN
			service_assign := FALSE;
			EXIT;
		ELSE
			service_assign := TRUE;
		END_IF
	END_IF
END_FOR

FOR idx_queue := 1 TO rs_count DO
	IF (i_service_req.request_cmd = TO_UINT(E_Util_Service_Req.Off))  THEN 
		IF  (service_req_queue[idx_queue].rs_number = i_service_req.rs_number)  THEN
			service_release := TRUE;
			EXIT;
		ELSE
			service_release := FALSE;
		END_IF
	END_IF
END_FOR


trig_service_assign(CLK := service_assign);
trig_service_release(CLK := service_release);


IF trig_service_assign.Q THEN
	FOR idx_queue := 1 TO rs_count DO
		IF i_rs_module_constrain THEN
			IF idx_queue = i_shared_rs THEN 
				rs_same_module := Check_RSs_SameModule(i_rs_1 := service_req_queue[idx_queue-1].rs_number, i_rs_2 := i_service_req.rs_number);
			ELSE
				rs_same_module := Check_RSs_SameModule(i_rs_1 := service_req_queue[idx_queue].rs_number, i_rs_2 := i_service_req.rs_number);
			END_IF
		END_IF
		IF service_req_queue[idx_queue].rs_number = i_service_req.rs_number THEN
			EXIT;
		ELSIF NOT service_req_queue[idx_queue].is_assigned AND  (service_req_queue[idx_queue].rs_number <> i_service_req.rs_number)  THEN 
				IF i_rs_module_constrain AND  (idx_queue = i_shared_rs) AND  rs_same_module THEN 
					CONTINUE;
				ELSE
					service_req_queue[idx_queue].is_assigned  := TRUE;
					service_req_queue[idx_queue].rs_number := i_service_req.rs_number;
					EXIT;
				END_IF
		END_IF
	END_FOR
END_IF



// Remove from queue
IF trig_service_release.Q THEN
	FOR idx_queue := 1 TO rs_count DO
		IF service_req_queue[idx_queue].rs_number =  i_service_req.rs_number THEN
			service_req_queue[idx_queue].rs_number := 0;
			service_req_queue[idx_queue].is_assigned  := FALSE;
			EXIT;
		END_IF
	END_FOR
END_IF

// Update queue

FOR idx_queue := 1 TO rs_count DO
	IF  NOT service_req_queue[idx_queue].is_assigned  THEN 
		FOR idx_queue_update := idx_queue + 1 TO rs_count DO
			IF i_rs_module_constrain THEN
				IF idx_queue = i_shared_rs THEN 
					rs_same_module := Check_RSs_SameModule(i_rs_1 := service_req_queue[idx_queue-1].rs_number, i_rs_2 := service_req_queue[idx_queue_update].rs_number);
				ELSE
					rs_same_module := Check_RSs_SameModule(i_rs_1 := service_req_queue[idx_queue].rs_number, i_rs_2 := service_req_queue[idx_queue_update].rs_number);
				END_IF
			END_IF
			IF service_req_queue[idx_queue_update].rs_number > 0 THEN 
				IF  NOT i_rs_module_constrain THEN 
					service_req_queue[idx_queue] := service_req_queue[idx_queue_update];
					service_req_queue[idx_queue_update].rs_number := 0;
					service_req_queue[idx_queue_update].is_assigned := FALSE;
					EXIT;
				ELSIF i_rs_module_constrain AND NOT (idx_queue = i_shared_rs) THEN 
					service_req_queue[idx_queue] := service_req_queue[idx_queue_update];
					service_req_queue[idx_queue_update].rs_number := 0;
					service_req_queue[idx_queue_update].is_assigned := FALSE;
					EXIT;
				ELSIF i_rs_module_constrain AND  (idx_queue = i_shared_rs) AND NOT rs_same_module THEN
					service_req_queue[idx_queue] := service_req_queue[idx_queue_update];
					service_req_queue[idx_queue_update].rs_number := 0;
					service_req_queue[idx_queue_update].is_assigned := FALSE;
					EXIT;
				ELSIF i_rs_module_constrain AND  (idx_queue = i_shared_rs) AND  rs_same_module THEN
					CONTINUE;				
				END_IF
			END_IF						
		END_FOR	
	END_IF
END_FOR

// Service on/off requet to Utilities

o_service_req := service_req_queue[1].is_assigned ; // on request to utilities if queue pos #1 is populated / has a RS assigned 


// Service assigned sts to RS controller

IF i_shared_rs >= 2 THEN
	FOR idx_queue := 1 TO i_shared_rs DO 
		IF service_req_queue[idx_queue].is_assigned THEN 
			o_assigned_rs_number[idx_queue] := service_req_queue[idx_queue].rs_number;
		ELSE
			o_assigned_rs_number[idx_queue] := 0;
		END_IF
	END_FOR
ELSIF i_shared_rs = 1 THEN
	IF service_req_queue[idx_queue].is_assigned THEN 
		o_assigned_rs_number[1] := service_req_queue[1].rs_number;
	ELSE
		o_assigned_rs_number[1] := 0;
	END_IF
END_IF

METHOD Check_RSs_SameModule : BOOL
VAR_INPUT
	i_rs_1 : UINT;
	i_rs_2 : UINT;
END_VAR

Check_RSs_SameModule := ((i_rs_1 >=1  AND i_rs_1 <= 3) AND (i_rs_2 >=1  AND i_rs_2 <= 3)) OR 
						((i_rs_1 >=4  AND i_rs_1 <= 6) AND (i_rs_2 >=4  AND i_rs_2 <= 6)) OR 
                        ((i_rs_1 >=7  AND i_rs_1 <= 9) AND (i_rs_2 >=7  AND i_rs_2 <= 9)) OR
						((i_rs_1 >=10 AND i_rs_1<= 12) AND (i_rs_2 >=10 AND i_rs_2 <= 12));
END_METHOD

METHOD Clear_Queue : BOOL
VAR_INPUT
END_VAR
FOR idx_queue := 1 TO rs_count DO
	service_req_queue[idx_queue].rs_number := 0;
	service_req_queue[idx_queue].is_assigned  := FALSE;
END_FOR
END_METHOD

END_FUNCTION_BLOCK

// ---- Function_Blocks/FB_SetOutput_TwoInputs.TcPOU
FUNCTION_BLOCK FB_SetOutput_TwoInputs
VAR_IN_OUT
	io_in1 	: REAL;
	io_in2	: REAL;
END_VAR
VAR_OUTPUT
	o_set_value : REAL;
END_VAR
VAR
	in1_changed : BOOL;
	in2_changed : BOOL;
	
	in1_prev : REAL;
	in2_prev : REAL;
	
	in_latest : REAL;
END_VAR

// Rising edge detection for Input1
in1_changed := (io_in1 <> in1_prev ) ;
// Rising edge detection for Input2
in2_changed := (io_in2 <> in2_prev ) ;

// Determine which input has a rising edge
IF in1_changed THEN
	in1_prev 	:= io_in1;
    in_latest 	:= io_in1;
	io_in2 		:= in_latest;
ELSIF in2_changed THEN	
	in2_prev 	:= io_in2;
    in_latest 	:= io_in2;
	io_in1 		:= in_latest;
END_IF


// Set the output to the latest input
o_set_value := in_latest;

END_FUNCTION_BLOCK

// ---- Function_Blocks/FB_Utilities_Service.TcPOU
FUNCTION_BLOCK FB_Utilities_Service
VAR_INPUT
	i_service_req : ST_Util_Service_Req;
	
END_VAR
VAR_OUTPUT
	o_service_sts 	: ST_Util_Service_Sts;
END_VAR
VAR
	in_service_sts 			AT %I* : BYTE;
	in_service_error_code  	AT %I* : DWORD;
	
	out_service_req 		AT %Q* : BYTE;

END_VAR

out_service_req := TO_BYTE(i_service_req.request_cmd);


o_service_sts.idle 				:= in_service_sts = E_Util_Service_Sts.PowerUp;
o_service_sts.ready 			:= in_service_sts = E_Util_Service_Sts.Active;
o_service_sts.running 			:= in_service_sts = E_Util_Service_Sts.Running;
o_service_sts.faulted 			:= in_service_sts = E_Util_Service_Sts.Faulted;
o_service_sts.error_code		:= in_service_error_code;

END_FUNCTION_BLOCK
